TYPE Prozessvariablen :
STRUCT
	q1					:LREAL;				// X-Koordinate oder Gelenkwinkel 1
	q2					:LREAL;				// Y-Koordinate oder Gelenkwinkel 2
	q3					:LREAL;				// Z-Koordinate oder Gelenkwinkel 3
	q4					:LREAL;				// Orintierung um X-Achse oder Gelenkwinkel 4
	q5					:LREAL;				// Orientierung um Y-Achse oder Gelenkwinkel 5
	q6					:LREAL;				// Orientierung um Z-Achse oder Gelenkwinkel 6
	v					:LREAL;				// Geschwindigkeit
	a					:LREAL;				// Beschleunigung
	PosTyp				:Positionsart;		// Position-Typ definieren (Absolut / Relativ)		
	MoveTyp				:Bewegungsart;		// Bewegungsart definieren (Linear / Circular etc.)
END_STRUCT
END_TYPE

(* stored: Version 1.1.0.1
   DUT Prozessvariablen: Id {49970fae-9394-400d-bf68-faab23befb20} *)
